// TIA Portal V21 export
DATA_BLOCK "Alarms_DB"   // DB201
{ S7_Optimized_Access := 'FALSE'; DB_Accessible_From_OPC_UA := 'FALSE' }
// stored: AutoNumber false, DBAccessibleFromOPCUA false, DBAccessibleFromWebserver false
   VAR
      General { ExternalWritable := 'False'} : Struct
         EmergencyStop : Bool;
      END_STRUCT;
      PLC { ExternalWritable := 'False'} : Struct
         SupplyModule2 : Bool;
         SupplyModule3 : Bool;
         SupplyModule4 : Bool;
         SupplyModule5 : Bool;
         FeedbackModule2 : Bool;
         FeedbackModule3 : Bool;
         FeedbackModule4 : Bool;
         FeedbackModule5 : Bool;
      END_STRUCT;
      Sensors { ExternalWritable := 'False'} : Struct
         TankLevel1_Wiring : Bool;
         TankLevel2_Wiring : Bool;
      END_STRUCT;
      Pumps { ExternalWritable := 'False'} : Struct
         CircuitProtection_1 : Bool;
         ContactorNotON_1 : Bool;
         ContactorNotOFF_1 : Bool;
         SoftstartNotON_1 : Bool;
         SoftstartNotBypassed_1 : Bool;
         SoftstartStuckBypassed_1 : Bool;
         SoftstartNotOFF_1 : Bool;
         SoftstartFault_1 : Bool;
         CircuitProtection_2 : Bool;
         ContactorNotON_2 : Bool;
         ContactorNotOFF_2 : Bool;
         SoftstartNotON_2 : Bool;
         SoftstartNotBypassed_2 : Bool;
         SoftstartStuckBypassed_2 : Bool;
         SoftstartNotOFF_2 : Bool;
         SoftstartFault_2 : Bool;
      END_STRUCT;
   END_VAR
BEGIN
END_DATA_BLOCK
